(* IEC 61131-3 sources: motion-control-precision-force/07-codesys-fb, 7 files *)

(* ---- DUT_ServoAI_Params.st ---- *)
// ================================================================
// DUT_ServoAI_Params — AI Servo Parameter Structure
// ================================================================
// Central parameter struct for all servo AI function blocks.
// Parameters are trained offline (PPO/LightGBM/linear regression)
// and written to this struct via Modbus TCP or CODESYS recipe.
//
// To update: edge IPC trains new model → writes to PLC holding
// registers → CODESYS copies to this struct → FB uses new params.
// ================================================================

TYPE DUT_ServoAI_Params :
STRUCT
    // ============================================================
    // FB_ForceControl — Force control parameters
    // ============================================================
    rForce_Kp         : REAL := 0.5;
    rForce_Ki         : REAL := 0.02;
    rForce_Kd         : REAL := 0.0;
    iForce_ContactThr : INT  := 50;    // Contact threshold (‰)
    iForce_MaxTorque  : INT  := 800;   // Safety max (‰)
    iForce_MaxTime    : UDINT := 5000; // Max hold time (ms)

    // ============================================================
    // FB_GainScheduler — Gain scheduling tables (4 zones)
    // ============================================================
    rGain_Z1_KpVel    : REAL := 40.0;
    rGain_Z1_KiVel    : REAL := 20.0;
    rGain_Z1_KpPos    : REAL := 30.0;
    rGain_Z1_Kff      : REAL := 0.0;

    rGain_Z2_KpVel    : REAL := 60.0;
    rGain_Z2_KiVel    : REAL := 30.0;
    rGain_Z2_KpPos    : REAL := 45.0;
    rGain_Z2_Kff      : REAL := 30.0;

    rGain_Z3_KpVel    : REAL := 80.0;
    rGain_Z3_KiVel    : REAL := 40.0;
    rGain_Z3_KpPos    : REAL := 60.0;
    rGain_Z3_Kff      : REAL := 50.0;

    rGain_Z4_KpVel    : REAL := 35.0;
    rGain_Z4_KiVel    : REAL := 15.0;
    rGain_Z4_KpPos    : REAL := 25.0;
    rGain_Z4_Kff      : REAL := 60.0;

    rGain_SmoothFactor: REAL := 0.1;   // EMA smoothing

    // ============================================================
    // FB_ServoDiag — Diagnostic thresholds
    // ============================================================
    rDiag_CurW0       : REAL := 0.012;
    rDiag_CurW1       : REAL := 0.085;
    rDiag_CurBias     : REAL := 5.0;
    rDiag_CurRatioHi  : REAL := 1.30;
    rDiag_CurRatioLo  : REAL := 0.60;
    iDiag_FollErrLim  : DINT := 1000;
    iDiag_TempLim     : INT  := 850;
    iDiag_TempTrendLim: INT  := 50;

    // ============================================================
    // FB_ServoScope — Scope configuration
    // ============================================================
    iScope_TrigChannel : INT  := 1;
    rScope_TrigLevel   : REAL := 0.0;
    iScope_PreSamples  : INT  := 200;
    iScope_PostSamples : INT  := 800;

    // ============================================================
    // Meta
    // ============================================================
    sModelVersion     : STRING := 'v1.0.0';
    sModelDate        : STRING := '2026-06-04';
END_STRUCT
END_TYPE

(* ---- DUT_ServoDiag.st ---- *)
// ================================================================
// DUT_ServoDiag — Servo Diagnostic Data Structures
// ================================================================
// Auto-generated by AI Analyzer CodegenST
// Brand: delta-a3
// Author: AI Analyzer
// Generated: 2026-06-06 19:01
//
// ⚠ HITL PRINCIPLE: Parameter writes require operator authorization.
//    Set bAuthorized:=TRUE only after engineer confirms.
// ================================================================

/// Fault code enumeration
{attribute 'qualified_only'}
{attribute 'strict'}
TYPE E_ServoFault :
(
    eFault_None             := 0,
    eFault_CurrentSaturation := 1,
    eFault_SensorFault       := 2,
    eFault_FollowingError    := 3,
    eFault_OverTemp          := 4,
    eFault_MechanicalWear    := 5,
    eFault_DriveFault        := 6,
    eFault_Resonance         := 7,
    eFault_GainDeficiency    := 8,
    eFault_CurrentRipple     := 9,
    eFault_VelocityRipple    := 10
);
END_TYPE

/// HITL authorization state
TYPE E_HITLState :
(
    eHITL_Pending    := 0,  // Waiting for engineer feedback
    eHITL_Approved   := 1,  // Engineer authorized
    eHITL_Rejected   := 2,  // Engineer rejected
    eHITL_Delegated  := 3   // Delegated to another engineer
);
END_TYPE

/// Diagnostic session record (persistent)
TYPE ST_ServoSession :
STRUCT
    sSessionID      : STRING(36);   // UUID
    dtStartTime     : DT;           // Session start timestamp
    iTotalFaults    : UDINT;        // Cumulative fault count
    iAuthorizedCnt  : UDINT;        // Engineer-authorized actions
    iRejectedCnt    : UDINT;        // Engineer-rejected actions
    rAuthRate       : REAL;         // Authorization rate
END_STRUCT
END_TYPE

(* ---- FB_ForceControl.st ---- *)
// ================================================================
// FB_ForceControl — Closed-Loop Force/Torque Control for Dispensing
// ================================================================
// Implements precision force control for 3C dispensing applications.
// Uses CiA 402 CST (Cyclic Synchronous Torque) mode over EtherCAT.
//
// Control Modes:
//   0 = Idle
//   1 = Approach (position-controlled, fast)
//   2 = Contact Detect (torque threshold)
//   3 = Force Hold (PID force control)
//   4 = Retract
//
// Contact Detection:
//   Uses torque feedback spike to detect workpiece contact.
//   Threshold auto-adapted based on approach speed.
//
// Usage:
//   fbForce(
//     iActualTorque := %ID10,  // 0x6077 from PDO
//     iTargetForce  := 500,    // 5.00 N (scaled ×100)
//     bEnable       := TRUE
//   );
//   // Set iTorqueCommand (0x6071) to fbForce.iOutputTorque
// ================================================================

FUNCTION_BLOCK FB_ForceControl
VAR_INPUT
    // Feedback
    iActualTorque   : INT;      // 0x6077 Torque Actual Value (‰ rated)
    iActualPos      : DINT;     // 0x6064 Position Actual Value (pulses)

    // Setpoint
    iTargetForce    : INT;      // Target force (‰ rated torque, e.g. 500 = 50.0%)
    iApproachSpeed  : UDINT := 100000; // Approach speed (pulses/s)
    iRetractSpeed   : UDINT := 200000; // Retract speed (pulses/s)
    iRetractPos     : DINT;     // Position to retract to after dispensing

    // Tuning
    rForceKp        : REAL := 0.5;   // Force loop P gain
    rForceKi        : REAL := 0.02;  // Force loop I gain
    rForceKd        : REAL := 0.0;   // Force loop D gain
    iContactThreshold : INT := 50;   // Contact detection threshold (‰)
    iContactDebounce : INT := 5;     // Contact confirm cycles

    // Limits
    iMaxTorque      : INT  := 800;   // Safety: max torque (80%)
    iMaxForceTime   : UDINT := 5000; // Safety: max force hold time (ms)
    iPosLimitFwd    : DINT;          // Forward soft limit
    iPosLimitRev    : DINT;          // Reverse soft limit

    // Commands
    bStart          : BOOL;     // Rising edge: start dispensing cycle
    bStop           : BOOL;     // Rising edge: emergency stop
    bEnable         : BOOL;
END_VAR
VAR_OUTPUT
    iOutputTorque   : INT;      // 0x6071 Target Torque (‰ rated)
    iOutputMode     : SINT;     // 0x6060 Modes of Operation (10 = CST)
    iState          : INT;      // 0=Idle 1=Approach 2=Contact 3=Hold 4=Retract 5=Done 6=Fault
    bCycleComplete  : BOOL;     // Dispensing cycle finished
    bContactMade    : BOOL;     // Workpiece contact detected
    rForceActual    : REAL;     // Actual force (scaled)
    rForceError     : REAL;     // Force error
    iErrorCode      : INT;
END_VAR
VAR
    // State machine
    iPrevState      : INT;

    // Force PID
    rIntegral       : REAL;
    rPrevError      : REAL;
    rOutputRaw      : REAL;

    // Contact detection
    iContactCnt     : INT;
    rAvgTorqueBase  : REAL;     // Baseline torque (moving avg during approach)

    // Timing
    tHoldStart      : UDINT;
    tCurrent        : UDINT;

    // Edge detection
    bStartPrev      : BOOL;
    bStopPrev       : BOOL;
END_VAR

// ===== FB_ForceControl Method Body =====

IF NOT bEnable THEN
    iState := 0;
    iOutputTorque := 0;
    bCycleComplete := FALSE;
    RETURN;
END_IF;

// ── Safety: Emergency Stop ──
IF bStop AND NOT bStopPrev THEN
    iState := 6; // Fault
    iOutputTorque := 0;
    iErrorCode := 1;
END_IF;
bStopPrev := bStop;

// ── Start rising edge ──
IF bStart AND NOT bStartPrev AND iState = 0 THEN
    iState := 1; // Approach
    rIntegral := 0.0;
    rPrevError := 0.0;
    bCycleComplete := FALSE;
    bContactMade := FALSE;
    iContactCnt := 0;
    rAvgTorqueBase := 0.0;
END_IF;
bStartPrev := bStart;

// ── Current time (ms) ──
tCurrent := 0; // Placeholder — use PLC cycle counter or RTC in production

// ── State Machine ──
CASE iState OF
    // ────────────────────────────────────
    0: // Idle — waiting for start
        iOutputTorque := 0;
        iOutputMode := 8; // CSP mode for positioning

    // ────────────────────────────────────
    1: // Approach — fast positioning to workpiece
        iOutputMode := 8; // CSP mode
        iOutputTorque := 0;

        // Baseline torque tracking (moving avg for contact detection)
        rAvgTorqueBase := rAvgTorqueBase * 0.95 +
                          INT_TO_REAL(iActualTorque) * 0.05;

        // Contact detection: torque spike above baseline + threshold
        IF INT_TO_REAL(iActualTorque) > rAvgTorqueBase + INT_TO_REAL(iContactThreshold) THEN
            iContactCnt := iContactCnt + 1;
        ELSE
            iContactCnt := MAX(0, iContactCnt - 1);
        END_IF;

        IF iContactCnt >= iContactDebounce THEN
            iState := 2; // Contact confirmed
            bContactMade := TRUE;
        END_IF;

    // ────────────────────────────────────
    2: // Contact — transition to force control
        iOutputMode := 10; // CST mode
        rIntegral := 0.0;
        rPrevError := 0.0;
        tHoldStart := tCurrent;
        iState := 3; // Enter force hold

    // ────────────────────────────────────
    3: // Force Hold — PID force control
        iOutputMode := 10; // CST mode

        // Force error
        rForceActual := INT_TO_REAL(iActualTorque);
        rForceError  := INT_TO_REAL(iTargetForce) - rForceActual;

        // PID
        rIntegral := rIntegral + rForceError;
        // Anti-windup: clamp integral
        IF rIntegral > 500.0 THEN rIntegral := 500.0; END_IF;
        IF rIntegral < -500.0 THEN rIntegral := -500.0; END_IF;

        rOutputRaw := rForceKp * rForceError +
                      rForceKi * rIntegral +
                      rForceKd * (rForceError - rPrevError);
        rPrevError := rForceError;

        // Clamp output
        IF rOutputRaw > INT_TO_REAL(iMaxTorque) THEN
            rOutputRaw := INT_TO_REAL(iMaxTorque);
        END_IF;
        IF rOutputRaw < 0.0 THEN
            rOutputRaw := 0.0;
        END_IF;
        iOutputTorque := REAL_TO_INT(rOutputRaw);

        // Safety: force hold timeout
        IF (tCurrent - tHoldStart) > iMaxForceTime THEN
            iState := 4; // Timeout → retract
            iErrorCode := 2;
        END_IF;

        // Safety: position limit
        IF iActualPos > iPosLimitFwd OR iActualPos < iPosLimitRev THEN
            iState := 4; // Limit hit → retract
            iErrorCode := 3;
        END_IF;

    // ────────────────────────────────────
    4: // Retract — move back to safe position
        iOutputMode := 8; // CSP mode
        iOutputTorque := 0;
        // Check if retract complete (within window of target)
        IF ABS(iActualPos - iRetractPos) < 1000 THEN
            iState := 5; // Done
        END_IF;

    // ────────────────────────────────────
    5: // Done — cycle complete
        iOutputMode := 8;
        iOutputTorque := 0;
        bCycleComplete := TRUE;
        // Auto-reset to idle after one scan
        iState := 0;

    // ────────────────────────────────────
    6: // Fault
        iOutputTorque := 0;
        iOutputMode := 8;
        bCycleComplete := FALSE;

END_CASE;

(* ---- FB_GainScheduler.st ---- *)
// ================================================================
// FB_GainScheduler — Adaptive Servo Gain Scheduling
// ================================================================
// Automatically adjusts servo loop gains based on operating
// conditions (load, speed, position). Uses linear interpolation
// between pre-defined operating points.
//
// Operating Points (pre-configured — tuned offline with PPO/RL):
//   Low Load  (< 30% rated):  Conservative gains
//   Mid Load  (30-70%):       Standard gains
//   High Load (> 70% rated):  Aggressive gains
//   High Speed (> 80% max):   Reduced gains (stability)
//
// Outputs (to Delta A3 via SDO or PDO):
//   Velocity Loop Gain     (P1-04,  CoE 0x2104)
//   Velocity Loop Integral (P1-05,  CoE 0x2105)
//   Position Loop Gain     (P1-06,  CoE 0x2106)
//   Speed Feedforward      (P1-07,  CoE 0x2107)
//   Torque Filter          (P1-08,  CoE 0x2108)
//
// Usage: Call every servo cycle. Gains auto-adjust based on
// current load and speed feedback.
// ================================================================

FUNCTION_BLOCK FB_GainScheduler
VAR_INPUT
    // Feedback (from PDO)
    iActualCurrent  : INT;      // 0x6078 Current Actual Value (‰ rated)
    iActualSpeed    : DINT;     // 0x606C Velocity Actual Value (0.1 rpm)
    iActualPos      : DINT;     // 0x6064 Position Actual Value

    // Motor specs (for normalization)
    iRatedCurrent   : INT  := 1000;   // Rated current (‰, e.g. 1000 = 100%)
    iMaxSpeed       : DINT := 300000; // Max speed (0.1 rpm, e.g. 300000 = 3000 rpm)

    // ── Pre-configured operating point tables ──
    // Entries: [Load%, Speed%] → {Kp_vel, Ki_vel, Kp_pos, Kff, TorqFilt}

    // Zone 1: Low Load, Low Speed (< 30%, < 50%)
    rZ1_KpVel       : REAL := 40.0;
    rZ1_KiVel       : REAL := 20.0;
    rZ1_KpPos       : REAL := 30.0;
    rZ1_Kff         : REAL := 0.0;
    rZ1_TorqFilt    : REAL := 1.0;

    // Zone 2: Mid Load, Mid Speed (30-70%, 50-80%)
    rZ2_KpVel       : REAL := 60.0;
    rZ2_KiVel       : REAL := 30.0;
    rZ2_KpPos       : REAL := 45.0;
    rZ2_Kff         : REAL := 30.0;
    rZ2_TorqFilt    : REAL := 0.5;

    // Zone 3: High Load, Low-Mid Speed (> 70%, < 80%)
    rZ3_KpVel       : REAL := 80.0;
    rZ3_KiVel       : REAL := 40.0;
    rZ3_KpPos       : REAL := 60.0;
    rZ3_Kff         : REAL := 50.0;
    rZ3_TorqFilt    : REAL := 0.3;

    // Zone 4: High Speed, Any Load (> 80%)
    rZ4_KpVel       : REAL := 35.0;
    rZ4_KiVel       : REAL := 15.0;
    rZ4_KpPos       : REAL := 25.0;
    rZ4_Kff         : REAL := 60.0;
    rZ4_TorqFilt    : REAL := 0.2;

    // Interpolation config
    rSmoothFactor   : REAL := 0.1;  // 0.0=instant, 0.5=slow transition (EMA)
    iUpdateRate     : INT  := 10;   // Update every N cycles

    bEnable         : BOOL;
END_VAR
VAR_OUTPUT
    // Computed gains (write to Delta A3 parameters)
    rOutKpVel       : REAL;     // → P1-04 (0x2104)
    rOutKiVel       : REAL;     // → P1-05 (0x2105)
    rOutKpPos       : REAL;     // → P1-06 (0x2106)
    rOutKff         : REAL;     // → P1-07 (0x2107)
    rOutTorqFilt    : REAL;     // → P1-08 (0x2108)

    // Status
    rLoadPct        : REAL;     // Current load percentage
    rSpeedPct       : REAL;     // Current speed percentage
    iActiveZone     : INT;      // Active operating zone (1-4)
    bInTransition   : BOOL;     // TRUE during gain transition
END_VAR
VAR
    iCycleCnt       : INT;
    rLoadPrev       : REAL;
    rSpeedPrev      : REAL;
    // EMA-smoothed outputs
    rKpVel_ema      : REAL := 40.0;
    rKiVel_ema      : REAL := 20.0;
    rKpPos_ema      : REAL := 30.0;
    rKff_ema        : REAL := 0.0;
    rTfilt_ema      : REAL := 1.0;
END_VAR

// ===== FB_GainScheduler Method Body =====

IF NOT bEnable THEN
    RETURN;
END_IF;

// ── Cycle counter: don't update every scan ──
iCycleCnt := iCycleCnt + 1;
IF iCycleCnt < iUpdateRate THEN
    RETURN;
END_IF;
iCycleCnt := 0;

// ── Normalize load and speed to 0-100% ──
rLoadPct  := ABS(INT_TO_REAL(iActualCurrent)) / INT_TO_REAL(iRatedCurrent) * 100.0;
rSpeedPct := ABS(INT_TO_REAL(iActualSpeed))  / INT_TO_REAL(iMaxSpeed)    * 100.0;

// Clamp
IF rLoadPct  > 100.0 THEN rLoadPct  := 100.0; END_IF;
IF rSpeedPct > 100.0 THEN rSpeedPct := 100.0; END_IF;

// ── Determine operating zone ──
IF rSpeedPct > 80.0 THEN
    // Zone 4: High speed — stability priority
    iActiveZone := 4;
    rOutKpVel    := rZ4_KpVel;
    rOutKiVel    := rZ4_KiVel;
    rOutKpPos    := rZ4_KpPos;
    rOutKff      := rZ4_Kff;
    rOutTorqFilt := rZ4_TorqFilt;

ELSIF rLoadPct > 70.0 THEN
    // Zone 3: High load
    iActiveZone := 3;
    rOutKpVel    := rZ3_KpVel;
    rOutKiVel    := rZ3_KiVel;
    rOutKpPos    := rZ3_KpPos;
    rOutKff      := rZ3_Kff;
    rOutTorqFilt := rZ3_TorqFilt;

ELSIF rLoadPct > 30.0 THEN
    // Zone 2: Mid load
    iActiveZone := 2;
    rOutKpVel    := rZ2_KpVel;
    rOutKiVel    := rZ2_KiVel;
    rOutKpPos    := rZ2_KpPos;
    rOutKff      := rZ2_Kff;
    rOutTorqFilt := rZ2_TorqFilt;

ELSE
    // Zone 1: Low load
    iActiveZone := 1;
    rOutKpVel    := rZ1_KpVel;
    rOutKiVel    := rZ1_KiVel;
    rOutKpPos    := rZ1_KpPos;
    rOutKff      := rZ1_Kff;
    rOutTorqFilt := rZ1_TorqFilt;

END_IF;

// ── EMA smoothing — prevents gain jumps ──
rKpVel_ema  := rKpVel_ema  * (1.0 - rSmoothFactor) + rOutKpVel    * rSmoothFactor;
rKiVel_ema  := rKiVel_ema  * (1.0 - rSmoothFactor) + rOutKiVel    * rSmoothFactor;
rKpPos_ema  := rKpPos_ema  * (1.0 - rSmoothFactor) + rOutKpPos    * rSmoothFactor;
rKff_ema    := rKff_ema    * (1.0 - rSmoothFactor) + rOutKff      * rSmoothFactor;
rTfilt_ema  := rTfilt_ema  * (1.0 - rSmoothFactor) + rOutTorqFilt * rSmoothFactor;

rOutKpVel    := rKpVel_ema;
rOutKiVel    := rKiVel_ema;
rOutKpPos    := rKpPos_ema;
rOutKff      := rKff_ema;
rOutTorqFilt := rTfilt_ema;

bInTransition := ABS(rLoadPct - rLoadPrev) > 5.0 OR ABS(rSpeedPct - rSpeedPrev) > 5.0;
rLoadPrev  := rLoadPct;
rSpeedPrev := rSpeedPct;

(* ---- FB_ServoDiag.st ---- *)
// ================================================================
// FB_ServoDiag — Servo Drive Diagnostic Block
// ================================================================
// Auto-generated by AI Analyzer CodegenST
// Brand: delta-a3
// Author: AI Analyzer
// Generated: 2026-06-06 19:01
//
// ⚠ HITL PRINCIPLE: Parameter writes require operator authorization.
//    Set bAuthorized:=TRUE only after engineer confirms.
// ================================================================

FUNCTION_BLOCK FB_ServoDiag

VAR_INPUT
    // ── PDO Feedback (CiA 402) ──
    iActualPosition           : DINT   := 0;  // 0x6064 Position Actual Value
    iActualVelocity           : DINT   := 0;  // 0x606C Velocity Actual Value (0.1 rpm)
    iActualTorque             : INT    := 0;  // 0x6077 Torque Actual Value (permille rated)
    iActualCurrent            : INT    := 0;  // 0x6078 Current Actual Value (permille rated)
    iFollowingError           : DINT   := 0;  // 0x60F4 Following Error Actual Value
    iStatusWord               : UINT   := 0;  // 0x6041 Status Word
    iOpMode                   : INT    := 0;  // 0x6061 Modes of Operation Display
    iDigitalInputs            : UDINT  := 0;  // 0x60FD Digital Inputs

    // ── Detection Thresholds ──
    rCurrentSaturationThreshold : REAL := 200.0;  // current_saturation
    rCurrentWearThreshold : REAL := 112.0;  // current_wear
    rTrackingGainDeficiencyThreshold : REAL := 350.0;  // tracking_gain_deficiency
    rCurrentRippleThreshold : REAL := 10.5;  // current_ripple
    rVelocityRippleThreshold : REAL := 35.0;  // velocity_ripple

    // ── HITL Confirmation ──
    bOperatorConfirmed : BOOL := FALSE;  // Engineer authorization gate

    // ── Enable ──
    bEnable            : BOOL;
END_VAR
VAR_OUTPUT
    iFaultCode         : INT;      // 0=OK, see fault code table
    bAlarm             : BOOL;     // Any alarm active
    bShutdown          : BOOL;     // Critical fault -> E-Stop
    rFaultScore        : REAL;     // 0.0~1.0 confidence
    bCurrentSaturationDetected : BOOL;     // current_saturation
    bCurrentWearDetected : BOOL;     // current_wear
    bTrackingGainDeficiencyDetected : BOOL;     // tracking_gain_deficiency
    bCurrentRippleDetected : BOOL;     // current_ripple
    bVelocityRippleDetected : BOOL;     // velocity_ripple
END_VAR
VAR
    // ── Debounce counters ──
    iCurrentSaturationCnt     : INT := 0;
    iCurrentWearCnt     : INT := 0;
    iTrackingGainDeficiencyCnt     : INT := 0;
    iCurrentRippleCnt     : INT := 0;
    iVelocityRippleCnt     : INT := 0;

    // ── Constants ──
    iDebounceLimit     : INT := 10;  // Consecutive cycles to confirm
END_VAR

// ===== FB_ServoDiag Method Body =====

// ── Enable Gate ──
IF NOT bEnable THEN
    bAlarm    := FALSE;
    bShutdown := FALSE;
    iFaultCode := 0;
    RETURN;
END_IF;

// ── current_saturation: 250% saturation ──
IF INT_TO_REAL(iActualCurrent) > rCurrentSaturationThreshold THEN
    iCurrentSaturationCnt := iCurrentSaturationCnt + 1;
ELSE
    iCurrentSaturationCnt := MAX(0, iCurrentSaturationCnt - 1);
END_IF;

// ── current_wear: CUSUM drift 80->160% ──
IF INT_TO_REAL(iActualCurrent) > rCurrentWearThreshold THEN
    iCurrentWearCnt := iCurrentWearCnt + 1;
ELSE
    iCurrentWearCnt := MAX(0, iCurrentWearCnt - 1);
END_IF;

// ── tracking_gain_deficiency: Gain ratio 2.1x ──
IF ABS(INT_TO_REAL(iFollowingError)) > rTrackingGainDeficiencyThreshold THEN
    iTrackingGainDeficiencyCnt := iTrackingGainDeficiencyCnt + 1;
ELSE
    iTrackingGainDeficiencyCnt := MAX(0, iTrackingGainDeficiencyCnt - 1);
END_IF;

// ── current_ripple: HF ripple detected ──
IF INT_TO_REAL(iActualCurrent) > rCurrentRippleThreshold THEN
    iCurrentRippleCnt := iCurrentRippleCnt + 1;
ELSE
    iCurrentRippleCnt := MAX(0, iCurrentRippleCnt - 1);
END_IF;

// ── velocity_ripple: Velocity oscillation ──
IF INT_TO_REAL(iActualVelocity) > rVelocityRippleThreshold THEN
    iVelocityRippleCnt := iVelocityRippleCnt + 1;
ELSE
    iVelocityRippleCnt := MAX(0, iVelocityRippleCnt - 1);
END_IF;

// ── Fault Aggregation ──
iFaultCode := 0;
bAlarm     := FALSE;
bShutdown  := FALSE;
rFaultScore := 0.0;

IF iCurrentSaturationCnt >= iDebounceLimit THEN
    iFaultCode := 1;
    bAlarm     := TRUE;
    bShutdown  := TRUE;
    rFaultScore := MIN(1.0, INT_TO_REAL(iCurrentSaturationCnt) / 20.0);
    bCurrentSaturationDetected := TRUE;
ELSIF iCurrentWearCnt >= iDebounceLimit THEN
    iFaultCode := 2;
    bAlarm     := TRUE;
    bShutdown  := FALSE;
    rFaultScore := MIN(1.0, INT_TO_REAL(iCurrentWearCnt) / 20.0);
    bCurrentWearDetected := TRUE;
ELSIF iTrackingGainDeficiencyCnt >= iDebounceLimit THEN
    iFaultCode := 3;
    bAlarm     := TRUE;
    bShutdown  := FALSE;
    rFaultScore := MIN(1.0, INT_TO_REAL(iTrackingGainDeficiencyCnt) / 20.0);
    bTrackingGainDeficiencyDetected := TRUE;
ELSIF iVelocityRippleCnt >= iDebounceLimit THEN
    iFaultCode := 5;
    bAlarm     := TRUE;
    bShutdown  := FALSE;
    rFaultScore := MIN(1.0, INT_TO_REAL(iVelocityRippleCnt) / 20.0);
    bVelocityRippleDetected := TRUE;
ELSIF iCurrentRippleCnt >= iDebounceLimit THEN
    iFaultCode := 4;
    bAlarm     := TRUE;
    bShutdown  := FALSE;
    rFaultScore := MIN(1.0, INT_TO_REAL(iCurrentRippleCnt) / 20.0);
    bCurrentRippleDetected := TRUE;
END_IF;

// ── Reset detection flags ──
IF iFaultCode = 0 THEN
    bCurrentSaturationDetected := FALSE;
    bCurrentWearDetected := FALSE;
    bTrackingGainDeficiencyDetected := FALSE;
    bCurrentRippleDetected := FALSE;
    bVelocityRippleDetected := FALSE;
END_IF;

(* ---- FB_ServoScope.st ---- *)
// ================================================================
// FB_ServoScope — EtherCAT PDO Data Capture for Oscilloscope
// ================================================================
// Captures Cyclic PDO data from EtherCAT slaves into a PLC ring
// buffer array. Designed to feed an external oscilloscope (HMI,
// SCADA, or edge IPC via Modbus TCP).
//
// Captured Signals (from CiA 402 + Delta A3 CoE objects):
//   CH1: Position Actual Value   (0x6064)    — INT32
//   CH2: Velocity Actual Value   (0x606C)    — INT32
//   CH3: Current Actual Value    (0x6078)    — INT16
//   CH4: Torque Actual Value     (0x6077)    — INT16
//   CH5: Following Error         (0x60F4)    — INT32
//   CH6: Status Word             (0x6041)    — UINT16
//   CH7: Digital Inputs          (0x60FD)    — UINT32
//   CH8: Modes of Operation      (0x6061)    — INT8
//
// Buffer: 1000 samples × 8 channels, ring buffer (FIFO)
// Trigger: level trigger on any channel, rising/falling edge
//
// Usage:
//   fbScope(
//     iPosActual := %ID0,   // from PDO image
//     iVelActual := %ID4,
//     iCurActual  := %ID8,
//     ...
//     bEnable := TRUE
//   );
//   // Read captured data from fbScope.arBuffer
// ================================================================

FUNCTION_BLOCK FB_ServoScope
VAR_INPUT
    // PDO Inputs (mapped from EtherCAT I/O image)
    iPosActual      : DINT;     // 0x6064 Position Actual Value
    iVelActual      : DINT;     // 0x606C Velocity Actual Value
    iCurActual      : INT;      // 0x6078 Current Actual Value
    iTrqActual      : INT;      // 0x6077 Torque Actual Value
    iFollErr        : DINT;     // 0x60F4 Following Error Actual Value
    iStatusWord     : UINT;     // 0x6041 Status Word
    iDigInputs      : UDINT;    // 0x60FD Digital Inputs
    iOpMode         : SINT;     // 0x6061 Modes of Operation Display

    bEnable         : BOOL;     // Enable capture

    // Trigger config
    bTrigEnable     : BOOL;     // Enable trigger mode
    iTrigChannel    : INT  := 1; // Trigger source channel (1-8)
    rTrigLevel      : REAL := 0.0; // Trigger level
    bTrigEdge       : BOOL := TRUE; // TRUE=Rising, FALSE=Falling
    iTrigPreSamples : INT  := 200;  // Pre-trigger samples to retain
    iTrigPostSamples: INT  := 800;  // Post-trigger samples
END_VAR
VAR_OUTPUT
    // Ring buffer (exposed for HMI/SCADA readout)
    arBuffer        : ARRAY[0..7, 0..999] OF REAL;  // 8ch × 1000 samples
    iBufHead        : INT;      // Current write position (0..999)
    iBufCount       : UDINT;    // Total samples captured
    iBufSamples     : INT;      // Valid samples in buffer (0..1000)
    bBufFull        : BOOL;     // Buffer full (1000 samples)
    bTriggered      : BOOL;     // Trigger fired
    iTrigPosition   : INT;      // Buffer index of trigger point (-1 = none)

    // Status
    bActive         : BOOL;
    iErrorCode      : INT;
END_VAR
VAR
    bInit           : BOOL := TRUE;
    bArming         : BOOL;
    iPreCounter     : INT;
    iPostCounter    : INT;
    rPrevTrigVal    : REAL;
    arrChValues     : ARRAY[0..7] OF REAL;
    bTrigEdgePrev   : BOOL;
END_VAR

// ===== FB_ServoScope Method Body =====

IF NOT bEnable THEN
    bActive := FALSE;
    RETURN;
END_IF;

// ── Initialize buffer on first cycle ──
IF bInit THEN
    FOR i: INT := 0 TO 7 DO
        FOR j: INT := 0 TO 999 DO
            arBuffer[i, j] := 0.0;
        END_FOR;
    END_FOR;
    iBufHead    := 0;
    iBufCount   := 0;
    iBufSamples := 0;
    bBufFull    := FALSE;
    bTriggered  := FALSE;
    iTrigPosition := -1;
    bInit       := FALSE;
    bArming     := bTrigEnable;
    iPreCounter := iTrigPreSamples;
    iPostCounter:= 0;
END_IF;

bActive := TRUE;

// ── Assemble channel values ──
arrChValues[0] := INT_TO_REAL(iPosActual);
arrChValues[1] := INT_TO_REAL(iVelActual);
arrChValues[2] := INT_TO_REAL(iCurActual);
arrChValues[3] := INT_TO_REAL(iTrqActual);
arrChValues[4] := INT_TO_REAL(iFollErr);
arrChValues[5] := UINT_TO_REAL(iStatusWord);
arrChValues[6] := UDINT_TO_REAL(iDigInputs);
arrChValues[7] := SINT_TO_REAL(iOpMode);

// ── Trigger logic ──
IF bTrigEnable THEN
    IF iTrigChannel >= 1 AND iTrigChannel <= 8 THEN
        IF bArming THEN
            // Pre-trigger: fill buffer without marking trigger
            IF iPreCounter > 0 THEN
                iPreCounter := iPreCounter - 1;
            ELSE
                bArming := FALSE;
            END_IF;
        ELSE
            // Check trigger condition
            IF iTrigChannel >= 1 AND iTrigChannel <= 8 THEN
                rPrevTrigVal := arrChValues[iTrigChannel - 1];
                IF bTrigEdge THEN
                    // Rising edge
                    IF rPrevTrigVal < rTrigLevel AND
                       arrChValues[iTrigChannel - 1] >= rTrigLevel THEN
                        bTriggered := TRUE;
                        iTrigPosition := iBufHead;
                        iPostCounter := iTrigPostSamples;
                    END_IF;
                ELSE
                    // Falling edge
                    IF rPrevTrigVal > rTrigLevel AND
                       arrChValues[iTrigChannel - 1] <= rTrigLevel THEN
                        bTriggered := TRUE;
                        iTrigPosition := iBufHead;
                        iPostCounter := iTrigPostSamples;
                    END_IF;
                END_IF;
            END_IF;

            // Post-trigger countdown
            IF bTriggered AND iPostCounter > 0 THEN
                iPostCounter := iPostCounter - 1;
                IF iPostCounter = 0 THEN
                    bTrigEnable := FALSE; // Single-shot: disarm after capture
                END_IF;
            END_IF;
        END_IF;
    END_IF;
END_IF;

// ── Write to ring buffer ──
FOR i: INT := 0 TO 7 DO
    arBuffer[i, iBufHead] := arrChValues[i];
END_FOR;

iBufHead  := (iBufHead + 1) MOD 1000;
iBufCount := iBufCount + 1;

IF iBufSamples < 1000 THEN
    iBufSamples := iBufSamples + 1;
END_IF;
IF iBufHead = 0 THEN
    bBufFull := TRUE;
END_IF;

(* ---- FB_ServoTune.st ---- *)
// ================================================================
// FB_ServoTune — Servo Parameter Tuning Block
// ================================================================
// Auto-generated by AI Analyzer CodegenST
// Brand: delta-a3
// Author: AI Analyzer
// Generated: 2026-06-06 19:01
//
// ⚠ HITL PRINCIPLE: Parameter writes require operator authorization.
//    Set bAuthorized:=TRUE only after engineer confirms.
// ================================================================

FUNCTION_BLOCK FB_ServoTune

VAR_INPUT
    // ── HITL Authorization ──
    bAuthorized        : BOOL;   // Engineer must set TRUE to execute
    bExecute           : BOOL;   // Rising edge triggers parameter write

    // ── Enable ──
    bEnable            : BOOL;
END_VAR

VAR_OUTPUT
    bBusy              : BOOL;   // Parameter write in progress
    bDone              : BOOL;   // All parameters written successfully
    bError             : BOOL;   // Write error
    iErrorID           : INT;    // SDO abort code (0 = OK)
    iParamIndex        : INT;    // Current parameter being written (0-based)
END_VAR

VAR
    // ── State machine ──
    iStep              : INT := 0;
    iStepCount         : INT := {len(recs)};

    // ── Edge detection ──
    bExecutePrev       : BOOL;
    bExecuteRising     : BOOL;

    // ── Target values ──
    rParam00X610B       : REAL := 320.0;
    rParam10X60Fb       : REAL := 0.0;
    rParam20X60A4       : REAL := 0.0;
    rParam30X6086       : REAL := 3.0;
END_VAR

// ===== FB_ServoTune Method Body =====

// ── Edge detection on bExecute ──
bExecuteRising := bExecute AND NOT bExecutePrev;
bExecutePrev   := bExecute;

// ── State Machine ──
CASE iStep OF

0:  // ── Idle: wait for authorization + execute trigger ──
    bBusy  := FALSE;
    bDone  := FALSE;
    bError := FALSE;
    IF bAuthorized AND bExecuteRising THEN
        iStep := 10;
    END_IF;

10:  // ── Write 0x610B: set (target: see rParam00X610B) ──
    bBusy := TRUE;
    iParamIndex := 0;
    // Resonance at 320Hz
    // SAFETY: Start with Q=0.5
    // TODO: Call vendor-specific SDO write FB for 0x610B
    // Example: fbSdoWrite(xExecute:=TRUE, iIndex:=24843, iSubIndex:=0, rValue:=rParam00X610B);
    iStep := 11;

11:  // ── Write 0x60FB: increase (target: see rParam10X60Fb) ──
    bBusy := TRUE;
    iParamIndex := 1;
    // Gain deficiency
    // SAFETY: Watch oscillation
    // TODO: Call vendor-specific SDO write FB for 0x60FB
    // Example: fbSdoWrite(xExecute:=TRUE, iIndex:=24827, iSubIndex:=0, rValue:=rParam10X60Fb);
    iStep := 12;

12:  // ── Write 0x60A4: decrease (target: see rParam20X60A4) ──
    bBusy := TRUE;
    iParamIndex := 2;
    // Velocity ripple
    // SAFETY: Check cycle time
    // TODO: Call vendor-specific SDO write FB for 0x60A4
    // Example: fbSdoWrite(xExecute:=TRUE, iIndex:=24740, iSubIndex:=0, rValue:=rParam20X60A4);
    iStep := 13;

13:  // ── Write 0x6086: set (target: see rParam30X6086) ──
    bBusy := TRUE;
    iParamIndex := 3;
    // Enable S-curve
    // TODO: Call vendor-specific SDO write FB for 0x6086
    // Example: fbSdoWrite(xExecute:=TRUE, iIndex:=24710, iSubIndex:=0, rValue:=rParam30X6086);
    iStep := 99;

99: // ── Done ──
    bBusy  := FALSE;
    bDone  := TRUE;
    iStep  := 0;

END_CASE;
